// Brief: Master Arm Test
FUNCTION_BLOCK PUBLIC FB_StateCtrlResponseTest EXTENDS FB_MasterArmCtrlBase
VAR_INPUT
END_VAR
VAR_OUTPUT
END_VAR
VAR
	//frequency test flag	
	m_freqTestFlag :ARRAY[1..7] OF BOOL;

	//step test flag
	m_stepTestFlag :ARRAY[1..7] OF BOOL;

	//init joint position
	m_initJntPos :Vec7d;
	
	//joint motion frequency
	m_jntMotionFreq :Vec7d :=[0.2, 0.2, 0.1, 4(0.1)];
	
	//joint motion range
	m_jntMotionRange :Vec7d :=[pi/6, pi/6, 0.1, 4(pi/6)];
	
	//test joint id
	m_testJntIdx :INT :=1;
	
	//step test joint angle
	m_jntStep : LREAL := 3*g_deg2Rad;
	
	//arm test step
	m_stepCycle:LREAL:=5;
	
	//timer
	m_time:LREAL;
	
	//step test direction
	m_stepTestDir :ARRAY[1..7] OF INT:=[1,1,1,1,1,1,1];
	
	//cycle time
	m_cycleTime:LREAL:=5;
	
	//parameters init flag
	m_paramInitFlag:BOOL;
	
	//test step
	m_testStep:INT:=-1;
	
	//start motion flag
	m_startMotion,m_startMotionLast:BOOL;
	
	//arm id
	m_armId:INT;
	
	//current DH joint position
	m_curDHJntPos:Vec7d;
	
	//basic function
	m_basicFun:FB_BasicFun;
	
	//DH joint position/velocity/acc
	m_cmdDHJntPos : VEC7d;
	m_cmdDHJntVel : VEC7d;
END_VAR

METHOD armJntTest : BOOL
VAR_INPUT
	i_masterArm :FB_MasterArm;
END_VAR

VAR
	
END_VAR


CASE m_testStep OF 
	0: //init the parameters
		m_freqTestFlag:=g_responseTest.m_freqTestFlag;
		m_stepTestFlag:=g_responseTest.m_stepTestFlag;		
		m_jntMotionFreq:=g_responseTest.m_jntMotionFreq;
		m_jntMotionRange:=g_responseTest.m_jntMotionRange;		
		m_jntStep:=g_responseTest.m_jntStep;		
		m_testJntIdx:=g_responseTest.m_testJntIdx;
		m_stepCycle:=g_responseTest.m_stepCycle;
				
		m_basicFun.activeJnt2DH(i_activeJntPos:= i_masterArm.curJntPos, o_DHJntPos=> m_curDHJntPos);
		//m_initJntPos := i_masterArm.curJntPos;
		m_initJntPos := m_curDHJntPos;
		m_jntOPMode := g_allPosMode;
		
		//after change the control mode,we need to change the inital target joint position and velocity
		m_cmdJntPos:=i_masterArm.curJntPos;
		m_cmdJntVel:=g_zeroVec7d;	
		m_cmdDHJntPos:=m_curDHJntPos;
		m_cmdDHJntVel:=g_zeroVec7d;
		m_time:=0;
		
		IF (m_testJntIdx >=1 AND m_testJntIdx <=7) THEN
			m_testStep:=10;
		END_IF
		
		
	10:// start the motion
		m_time:=m_time+g_armCtrlCycleTime;
		m_basicFun.activeJnt2DH(i_activeJntPos:= i_masterArm.curJntPos, o_DHJntPos=> m_curDHJntPos);
		
		IF (m_freqTestFlag[m_testJntIdx]=TRUE) AND (m_stepTestFlag[m_testJntIdx]=FALSE) THEN 
			m_cmdDHJntPos[m_testJntIdx]:=m_initJntPos[m_testJntIdx]+m_jntMotionRange[m_testJntIdx]/2
										+0.5*m_jntMotionRange[m_testJntIdx]*SIN(2*pi*m_jntMotionFreq[m_testJntIdx]*m_time-pi/2);
			m_cmdDHJntVel[m_testJntIdx]:=0.5*m_jntMotionRange[m_testJntIdx]*2*pi*m_jntMotionFreq[m_testJntIdx]*COS(2*pi*m_jntMotionFreq[m_testJntIdx]*m_time-pi/2);
		END_IF
		
		//step test
		IF (m_stepTestFlag[m_testJntIdx]=TRUE) AND (m_freqTestFlag[m_testJntIdx]=FALSE) THEN
			IF (m_time>m_cycleTime) THEN				
				//update the position every cycle
				m_time:=0;
				
				//change the joint motion direction
				IF (m_stepTestDir[m_testJntIdx]=1) THEN
					m_stepTestDir[m_testJntIdx]:=-1;
				ELSE
					m_stepTestDir[m_testJntIdx]:=1;
				END_IF
				
				//update the target joint position
				m_cmdDHJntPos[m_testJntIdx]:=m_initJntPos[m_testJntIdx]+0.5*m_jntStep*m_stepTestDir[m_testJntIdx];
				m_cmdDHJntVel[m_testJntIdx]:=0;			
			END_IF	
		END_IF
		
		//transform to active joint position		
		m_basicFun.DH2activeJnt(i_DHJntPos:=m_cmdDHJntPos, o_activeJntPos=> m_cmdJntPos);
		m_cmdJntVel:=m_cmdDHJntVel;
		
		//finish the test
		IF (m_startMotion=FALSE) THEN
			m_testStep:=20;
		END_IF
		
		
	20://finish signal
		m_testStep:=-1;
		
	
	-1: //
END_CASE
END_METHOD

METHOD PROTECTED calcCmdJntPos : BOOL
VAR_IN_OUT CONSTANT
	i_slaveIdx :INT;
	i_shoulderPose :ST_Frame;
	i_masterArm :FB_MasterArm;
	i_slaveStatus :ST_SlaveStatus;
END_VAR

VAR 
	errThres :LREAL;
	m_masterGripAngle: INT;
	i:int;
END_VAR

//init parameters flag
m_startMotion:=g_responseTest.m_startMotion[m_armId];

IF (m_startMotionLast=FALSE) AND (m_startMotion=TRUE)THEN
	m_testStep:=0;
END_IF
m_startMotionLast:=m_startMotion;

//frequency test and step test
armJntTest(i_masterArm);
END_METHOD

// override this function in each exact controller
METHOD PROTECTED calcCmdJntTrq : BOOL

VAR_IN_OUT CONSTANT
	i_slaveIdx :INT;
	i_shoulderPose :ST_Frame;
	i_masterArm :FB_MasterArm;
	i_slaveStatus :ST_SlaveStatus;
END_VAR

VAR 
	i:int;
END_VAR
m_cmdJntTrq:=g_zeroVec7d;
FOR i:=1 TO g_mJntNum DO 
	//m_cmdJntTrq[i] := m_cmdJntTrq[i] + i_masterArm.jntFriction[i] ;
END_FOR
END_METHOD

METHOD PUBLIC init : BOOL
VAR_IN_OUT CONSTANT
	i_masterArm	:FB_MasterArm;
END_VAR
VAR_IN_OUT 
	r_masterArmCtrlCmd :ST_ArmCtrlCmds;
END_VAR
// check if to hold the command joint position unchanged
m_holdLastCmds := checkToHoldLastCmds(i_masterArm);

// init
SUPER^.Init(i_masterArm,r_masterArmCtrlCmd);

// update commands to arm
copyCmds(r_masterArmCtrlCmd);

//init
m_startMotionLast:=FALSE;
m_armId:=i_masterArm.armIdx;
END_METHOD

END_FUNCTION_BLOCK

(* stored: Version 1.1.0.1, ProductVersion 3.1.4024.11
   POU FB_StateCtrlResponseTest: Id {de6669a5-1fe2-4852-8f76-c24f148c0802}, SpecialFunc None
   Method armJntTest: Id {7b22de9c-7f09-4d4d-b2c8-78a95b07f7f3}
   Method calcCmdJntPos: Id {57af1bb7-7499-481b-bb6b-1f8fc4340402}
   Method calcCmdJntTrq: Id {d58d17c1-a945-4533-a795-abb65c1d06cb}
   Method init: Id {3ff9d01f-3a1f-4163-b69f-dc2d88b2d932} *)
